(* IEC 61131-3 sources: CodesysTest/export/UN00 - Sharp Bagger/EM01 - Bagger Head/CM03 - Sealer/Electric/FB_SealWire.pou, 1 file *)

(* ---- FB_SealWire.pou.st ---- *)
(*#-#-#-#-#-#-#-#-#-#---Declaration---#-#-#-#-#-#-#-#-#-#-#-#-#*)

FUNCTION_BLOCK FINAL FB_SealWire EXTENDS FB_BasicSealer
VAR_INPUT
END_VAR
VAR_OUTPUT
	sealWireOutput : BOOL;
END_VAR
VAR

END_VAR
(*#-#-#-#-#-#-#-#-#-#---Implementation---#-#-#-#-#-#-#-#-#-#-#-#-#*)

SUPER^();
_stateString := TO_STRING(state);
IF sealActive THEN
	sealWireOutput := TRUE;
ELSE
	sealWireOutput := FALSE;
END_IF
